TYPE ST_Vis_OperationalControl :
STRUCT
	bVisInvisibleButton	: BOOL;	
	bVisInvisible		: BOOL;
	nFramePositionX		: REAL;
	nFramePositionY		: REAL;
	nButtonPositionX	: INT;
	nButtonPositionY	: INT;	
	
	bStartButtunState	: BOOL;
	bStopButtonState	: BOOL;
	bQuitButtonState	: BOOL;
	bEStopButtonState	: BOOL;
	
	bStartButtonLamp	: BOOL;
	bStopButtonLamp		: BOOL;
	bQuitButtonLamp		: BOOL;
	bEStopButtonLamp	: BOOL;
	
	bMessageColorGreen	: BOOL;
	bMessageColorRed	: BOOL;
	
	sMessage			: STRING;
	
	
END_STRUCT
END_TYPE

(* stored: Version 1.1.0.1, ProductVersion 3.1.4024.9
   DUT ST_Vis_OperationalControl: Id {38eeac75-11ec-4ffc-8d2d-cc762ea0111e} *)
